// TIA Portal V15.1 export
// export: Created 2024-06-21T08:40:46.8517399Z, ExportSetting WithDefaults, DisplayName Totally Integrated Automation Portal, DisplayVersion V15.1 Update 5, DisplayName TIA Portal Openness, DisplayVersion V15.1 Update 5, DisplayName SINAMICS Startdrive Advanced, DisplayVersion V15.1, DisplayName G130, G150, S120, S150, SINAMICS MV, S210, DisplayVersion V15.1, DisplayName G110M, G120, G120C, G120D, G120P, DisplayVersion V15.1, DisplayName STEP 7 Professional, DisplayVersion V15.1 Update 5, DisplayName STEP 7 Safety, DisplayVersion V15.1, DisplayName WinCC Professional, DisplayVersion V15.1 Update 5, DisplayName SIMATIC Visualization Architect, DisplayVersion V15.1
DATA_BLOCK "_209220ZS01Safety"   // DB375
{ S7_Optimized_Access := 'FALSE' }
VERSION : 0.1
// stored: AutoNumber false, DBAccessibleFromOPCUA true, IsOnlyStoredInLoadMemory false, IsWriteProtectedInAS false
   VAR RETAIN
      AA_209220AS10F9SH1 { ExternalAccessible := 'False'; ExternalVisible := 'False'; ExternalWritable := 'False'} : Bool;   // Emergency Stop push button 220AS10 (Operator panel)
      AA_209220AS11F9SH1 { ExternalAccessible := 'False'; ExternalVisible := 'False'; ExternalWritable := 'False'} : Bool;   // Emergency Stop push button 220AS11 (Operator panel)
      AA_209220AS20F9SH1 { ExternalAccessible := 'False'; ExternalVisible := 'False'; ExternalWritable := 'False'} : Bool;   // Emergency Stop push button 220AS20 (Start/Stop panel)
      AA_209220AS40F9SH1 { ExternalAccessible := 'False'; ExternalVisible := 'False'; ExternalWritable := 'False'} : Bool;   // Emergency Stop push button 220AS40 (External panel)
      AA_209220ASH01F9SH1 { ExternalAccessible := 'False'; ExternalVisible := 'False'; ExternalWritable := 'False'} : Bool;   // Emergency Stop push button 220ASH01 (Handheld panel)
      AA_209220ASH01F9SH2 { ExternalAccessible := 'False'; ExternalVisible := 'False'; ExternalWritable := 'False'} : Bool;   // Deathmans switch 220ASH01 (Handheld panel)
      AA_209000AK04F9QC1FB { ExternalAccessible := 'False'; ExternalVisible := 'False'; ExternalWritable := 'False'} : Bool;   // Feedback Alarm Contactor Brake 400VAC OFF 220CR21
      AA_209000AK04F9QC2FB { ExternalAccessible := 'False'; ExternalVisible := 'False'; ExternalWritable := 'False'} : Bool;   // Feedback Alarm Contactor Brake 400VAC OFF 220CR21
      AA_209000AK04F9QC3FB { ExternalAccessible := 'False'; ExternalVisible := 'False'; ExternalWritable := 'False'} : Bool;   // Feedback Alarm Contactor Brake 400VAC OFF 220CS22
      AA_209000AK04F9QC4FB { ExternalAccessible := 'False'; ExternalVisible := 'False'; ExternalWritable := 'False'} : Bool;   // Feedback Alarm Contactor Brake 400VAC OFF 220CS22
      AA_209000AK04F9QC5FB { ExternalAccessible := 'False'; ExternalVisible := 'False'; ExternalWritable := 'False'} : Bool;   // Feedback Alarm Contactor Brake 400VAC OFF 220CR23
      AA_209000AK04F9QC6FB { ExternalAccessible := 'False'; ExternalVisible := 'False'; ExternalWritable := 'False'} : Bool;   // Feedback Alarm Contactor Brake 400VAC OFF 220CR23
      AA_209220AS20XS10 { ExternalAccessible := 'False'; ExternalVisible := 'False'; ExternalWritable := 'False'} : Bool;   // Dummy plug is missing, no Handheld is connected 220AS20 (Start/Stop panel)
      AC_209220CS22M4SG10F { ExternalAccessible := 'False'; ExternalVisible := 'False'; ExternalWritable := 'False'} : Bool;   // Body present buth the safety sensor is not activated 220CS22M410F
      AC_209220CS22M4SG11F { ExternalAccessible := 'False'; ExternalVisible := 'False'; ExternalWritable := 'False'} : Bool;   // Body present buth the safety sensor is not activated 220CS22M411F
      "AC_209000AK04M1-UE140PSC-1" { ExternalAccessible := 'False'; ExternalVisible := 'False'; ExternalWritable := 'False'} : Bool;   // Position speed control - The infeed roller is busy with a tranfer to the slat conveyor but the slat conveyor is not running/too slow
      "AC_209000AK04M4-UE141PSC-1" { ExternalAccessible := 'False'; ExternalVisible := 'False'; ExternalWritable := 'False'} : Bool;   // Position speed control - The slat conveyor is busy with a tranfer to the outfeed roller but the outfeed roller is not running/too slow
      AA_209220ZS01SafetNotReseted { ExternalAccessible := 'False'; ExternalVisible := 'False'; ExternalWritable := 'False'} : Bool;   // Safety not Reseted 220ZS01
      AD_209220ZS01EmergencyStop { ExternalAccessible := 'False'; ExternalVisible := 'False'; ExternalWritable := 'False'} : Bool;   // Emergency Stop 220ZS01
      AD_209220ZS01GateStop { ExternalAccessible := 'False'; ExternalVisible := 'False'; ExternalWritable := 'False'} : Bool;   // Gate Stop 220ZS01
      AD_209220ZS01FbkError { ExternalAccessible := 'False'; ExternalVisible := 'False'; ExternalWritable := 'False'} : Bool;   // Feedback Error Pilz/Contactor 220ZS01
      AD_209220ZS01EStopPLC212 { ExternalAccessible := 'False'; ExternalVisible := 'False'; ExternalWritable := 'False'} : Bool;   // Emergency Stop from PLC212
      AD_209220ZS01MStopPLC212 { ExternalAccessible := 'False'; ExternalVisible := 'False'; ExternalWritable := 'False'} : Bool;   // Motion Stop from PLC212 for roller 220CR21
      AD_209220ZS01EStopPLC308 { ExternalAccessible := 'False'; ExternalVisible := 'False'; ExternalWritable := 'False'} : Bool;   // Emergency Stop from PLC318
      AD_209220ZS01MStopPLC308 { ExternalAccessible := 'False'; ExternalVisible := 'False'; ExternalWritable := 'False'} : Bool;   // Motion Stop from PLC318 for roller 220CR21
      "220AS10F9SH1AlarmABCondition" { ExternalAccessible := 'False'; ExternalVisible := 'False'; ExternalWritable := 'False'} : Bool;   // Alarm AB Condition
      "220AS11F9SH1AlarmABCondition" { ExternalAccessible := 'False'; ExternalVisible := 'False'; ExternalWritable := 'False'} : Bool;   // Alarm AB Condition
      "220AS20F9SH1AlarmABCondition" { ExternalAccessible := 'False'; ExternalVisible := 'False'; ExternalWritable := 'False'} : Bool;   // Alarm AB Condition
      "220AS40F9SH1AlarmABCondition" { ExternalAccessible := 'False'; ExternalVisible := 'False'; ExternalWritable := 'False'} : Bool;   // Alarm AB Condition
      "220ASH01F9SH1AlarmABCondition" { ExternalAccessible := 'False'; ExternalVisible := 'False'; ExternalWritable := 'False'} : Bool;   // Alarm AB Condition
      "220ASH01F9SH2AlarmABCondition" { ExternalAccessible := 'False'; ExternalVisible := 'False'; ExternalWritable := 'False'} : Bool;   // Alarm AB Condition
      "220AS20XS10AlarmABCondition" { ExternalAccessible := 'False'; ExternalVisible := 'False'; ExternalWritable := 'False'} : Bool;   // Alarm AB Condition
      AK04F9QC1FBAlarmABCondition { ExternalAccessible := 'False'; ExternalVisible := 'False'; ExternalWritable := 'False'} : Bool;   // Alarm AB Condition
      AK04F9QC2FBAlarmABCondition { ExternalAccessible := 'False'; ExternalVisible := 'False'; ExternalWritable := 'False'} : Bool;   // Alarm AB Condition
      AK04F9QC3FBAlarmABCondition { ExternalAccessible := 'False'; ExternalVisible := 'False'; ExternalWritable := 'False'} : Bool;   // Alarm AB Condition
      AK04F9QC4FBAlarmABCondition { ExternalAccessible := 'False'; ExternalVisible := 'False'; ExternalWritable := 'False'} : Bool;   // Alarm AB Condition
      AK04F9QC5FBAlarmABCondition { ExternalAccessible := 'False'; ExternalVisible := 'False'; ExternalWritable := 'False'} : Bool;   // Alarm AB Condition
      AK04F9QC6FBAlarmABCondition { ExternalAccessible := 'False'; ExternalVisible := 'False'; ExternalWritable := 'False'} : Bool;   // Alarm AB Condition
      SafetyNotResetedAlarmABCondition { ExternalAccessible := 'False'; ExternalVisible := 'False'; ExternalWritable := 'False'} : Bool;   // Alarm AB Condition
      H_209220AS10F9SH1IAnim : Word;   // Icon Animation
      H_209220AS11F9SH1IAnim : Word;   // Icon Animation
      H_209220AS20F9SH1IAnim : Word;   // Icon Animation
      H_209220AS40F9SH1IAnim : Word;   // Icon Animation
      H_209220ASH01F9SH1IAnim : Word;   // Icon Animation
      H_209220ASH01F9SH2IAnim : Word;   // Icon Animation
      H_209000AK04F9QC1FBIAnim : Word;   // Icon Animation
      H_209000AK04F9QC2FBIAnim : Word;   // Icon Animation
      H_209000AK04F9QC3FBIAnim : Word;   // Icon Animation
      H_209000AK04F9QC4FBIAnim : Word;   // Icon Animation
      H_209000AK04F9QC5FBIAnim : Word;   // Icon Animation
      H_209000AK04F9QC6FBIAnim : Word;   // Icon Animation
      H_209220AS20XS10IAnim : Word;   // Icon Animation
      H_209220CHB21M14SG1FIAnim : Word;   // Icon Animation
      H_209220CS22M4SG10FIAnim : Word;   // Icon Animation
      H_209220CS22M4SG11FIAnim : Word;   // Icon Animation
      H_209220ZS01SafetyNotResetedIAnim : Word;   // Icon Animation
      H_209220ZS01GateStopIAnim : Word;   // Icon Animation
      H_209220ZS01EmergencyStopIAnim : Word;   // Icon Animation
      H_209220ZS01FbkErrorIAnim : Word;   // Icon Animation
      H_209220ZS01EStopPLC212IAnim : Word;   // Icon Animation
      H_209220ZS01MStopPLC212IAnim : Word;   // Icon Animation
      H_209220ZS01EStopPLC308IAnim : Word;   // Icon Animation
      H_209220ZS01MStopPLC308IAnim : Word;   // Icon Animation
      H_209220ZS01PassivIAnim : Word;   // Icon Animation
      H_Anim : Word;   // Animation
      H_DBnr : Int;   // DB number
      Passivation { ExternalAccessible := 'False'; ExternalVisible := 'False'; ExternalWritable := 'False'} : "AlarmBits";   // Passivation Alarm Bits / Alarm A
      AlarmA { ExternalAccessible := 'False'; ExternalVisible := 'False'; ExternalWritable := 'False'} : Bool;   // Alarm A
      AlarmB { ExternalAccessible := 'False'; ExternalVisible := 'False'; ExternalWritable := 'False'} : Bool;   // Alarm B
      AlarmC { ExternalAccessible := 'False'; ExternalVisible := 'False'; ExternalWritable := 'False'} : Bool;   // Alarm C
      AlarmD { ExternalAccessible := 'False'; ExternalVisible := 'False'; ExternalWritable := 'False'} : Bool;   // Alarm D
      AlarmABCondition { ExternalAccessible := 'False'; ExternalVisible := 'False'; ExternalWritable := 'False'} : Bool;   // Summary Alarm AB condition
      SafetyObjectAckReq220AS10 { ExternalAccessible := 'False'; ExternalVisible := 'False'; ExternalWritable := 'False'} : Bool;   // Safety Status ACK REQ
      SafetyObjectAckReq220AS11 { ExternalAccessible := 'False'; ExternalVisible := 'False'; ExternalWritable := 'False'} : Bool;   // Safety Status ACK REQ
      SafetyObjectAckReq220AS20 { ExternalAccessible := 'False'; ExternalVisible := 'False'; ExternalWritable := 'False'} : Bool;   // Safety Status ACK REQ
      SafetyObjectAckReq220AS40 { ExternalAccessible := 'False'; ExternalVisible := 'False'; ExternalWritable := 'False'} : Bool;   // Safety Status ACK REQ
      SafetyObjectAckReq220ASH01 { ExternalAccessible := 'False'; ExternalVisible := 'False'; ExternalWritable := 'False'} : Bool;   // Safety Status ACK REQ
      PowerOnRequest { ExternalAccessible := 'False'; ExternalVisible := 'False'; ExternalWritable := 'False'} : Bool;   // Power On Request
      ResetSafetyActive { ExternalAccessible := 'False'; ExternalVisible := 'False'; ExternalWritable := 'False'} : Bool;   // Reset Safety Active
      FeedbackError { ExternalAccessible := 'False'; ExternalVisible := 'False'; ExternalWritable := 'False'} : Bool;   // Feedback Error
      Check220CS22M4SG10F { ExternalAccessible := 'False'; ExternalVisible := 'False'; ExternalWritable := 'False'} : Bool;   // Check if both safety sensors are activated
      Check220AS20XS10 { ExternalAccessible := 'False'; ExternalVisible := 'False'; ExternalWritable := 'False'} : Bool;   // Check if dummy plug is ok
   END_VAR
BEGIN
END_DATA_BLOCK
